// TwinCAT 3 PLC project PLC
// ProgramVersion: 3.1.4024.0
// CompilerDefines: MachineB
// libraries:
//   Tc2_Standard, * (Beckhoff Automation GmbH)
//   Tc2_System, * (Beckhoff Automation GmbH)
//   Tc3_Module, * (Beckhoff Automation GmbH)
// project tree:
//   Base/Datatype/ ST_Result.TcDUT
//   Base/FunctionBlock/ FB_Command.TcPOU
//   Base/Interface/ IBase.TcIO, ICommand.TcIO, IResult.TcIO
//   InterfaceBasics/DisplayExample/ FB_Display.TcPOU, FB_ProgressBar.TcPOU, IDisplay.TcIO
//   InterfaceBasics/SequenceExample/ FB_CylinderDoubleActing.TcPOU (not stored), FB_CylinderSequence.TcPOU, FB_CylinderSpringReturn.TcPOU (not stored), ICylinder.TcIO
//   InterfaceBasics/ PrgInterfaceBasics.TcPOU
//   / MAIN.TcPOU, PlcTask.TcTTO
// real-time tasks:
//   TASK PlcTask: cycle T#10ms, priority 20, ADS port 350

CONFIGURATION PLC
    RESOURCE PLC ON TwinCAT3
        TASK PlcTask(INTERVAL := T#10ms, PRIORITY := 20);
        PROGRAM MAIN WITH PlcTask : MAIN;
    END_RESOURCE
END_CONFIGURATION

// ---- Base/Datatype/ST_Result.TcDUT
{attribute 'pack_mode' := '1'}
TYPE ST_Result :
	STRUCT
		Busy	: BOOL;
		Error	: BOOL;
		Done	: BOOL;
		ErrorId : DINT;
	END_STRUCT
END_TYPE

// ---- Base/Interface/IBase.TcIO
INTERFACE IBase EXTENDS __System.IQueryInterface

END_INTERFACE

// ---- Base/Interface/ICommand.TcIO
INTERFACE ICommand EXTENDS IResult

PROPERTY Sequence : DINT
GET
END_GET
SET
END_SET
END_PROPERTY

METHOD Start : ICommand
VAR_INPUT
END_VAR
END_METHOD

END_INTERFACE

// ---- Base/Interface/IResult.TcIO
INTERFACE IResult EXTENDS __SYSTEM.IQueryInterface

PROPERTY Busy : BOOL
GET
END_GET
SET
END_SET
END_PROPERTY

PROPERTY Done : BOOL
GET
END_GET
SET
END_SET
END_PROPERTY

PROPERTY Error : BOOL
GET
END_GET
SET
END_SET
END_PROPERTY

PROPERTY ErrorId : DINT
GET
END_GET
SET
END_SET
END_PROPERTY

END_INTERFACE

// ---- InterfaceBasics/DisplayExample/IDisplay.TcIO
INTERFACE IDisplay EXTENDS IBase

METHOD Show : BOOL
VAR_INPUT
	Message : T_MaxString;
END_VAR
END_METHOD

END_INTERFACE

// ---- InterfaceBasics/SequenceExample/ICylinder.TcIO
INTERFACE ICylinder EXTENDS IBase

METHOD Extend : BOOL
VAR_INPUT
END_VAR
END_METHOD

METHOD Retract : BOOL
VAR_INPUT
END_VAR
END_METHOD

END_INTERFACE

// ---- MAIN.TcPOU
PROGRAM MAIN
VAR
END_VAR

PrgInterfaceBasics();

END_PROGRAM

// ---- InterfaceBasics/PrgInterfaceBasics.TcPOU
PROGRAM PrgInterfaceBasics
VAR
	// Interface Sequence Example
	{IF defined (MachineA)}
	CylinderSpringReturn : FB_CylinderSpringReturn;
	{ELSE}
	CylinderDoubleActing : FB_CylinderDoubleActing;
	{END_IF}
	CylinderSequence : FB_CylinderSequence;

	// Interface Display Example
	Display		 : FB_Display;
	ProgressBar	 : FB_ProgressBar;
	MainSequence : DINT := 0;
END_VAR

// Interface Sequence Example
{IF defined (MachineA)}

// Run Sequence with first Cylinder Type
CylinderSequence.Run(Cylinder := CylinderSpringReturn);
{ELSE}
CASE MainSequence OF
	0:
		IF CylinderSequence.Run(Cylinder := CylinderDoubleActing).Start().Busy THEN
			MainSequence := MainSequence + 10;
		END_IF

	10:
		IF CylinderSequence.Run(Cylinder := CylinderDoubleActing).Done THEN
			MainSequence := MainSequence + 10;
		END_IF

	20: // Next Command
END_CASE

{END_IF}

// Interface Display Example
ProgressBar.DisplayProgress(Display);

END_PROGRAM

// ---- InterfaceBasics/SequenceExample/FB_CylinderSequence.TcPOU
FUNCTION_BLOCK FB_CylinderSequence
VAR
	
END_VAR

METHOD PUBLIC Run : ICommand
VAR_INPUT
	Cylinder : ICylinder;
END_VAR

VAR_INST
	WaitTime : TON;
	Command	 : FB_Command;
END_VAR
IF Cylinder = 0 THEN
	Command.Error	:= TRUE;
	Command.ErrorId := 1;
	RETURN;
END_IF

CASE Command.Sequence OF
	0: // Extend
		IF Cylinder.Extend() THEN
			Command.Sequence := Command.Sequence + 10;
		END_IF

	10: // Wait 1s
		WaitTime.IN := TRUE;
		IF WaitTime.Q THEN
			WaitTime.IN		 := FALSE;
			Command.Sequence := Command.Sequence + 10;
		END_IF

	20: // Retract
		IF Cylinder.Retract() THEN
			Command.Sequence := Command.Sequence + 10;
		END_IF

	30: // Wait 1s
		WaitTime.IN := TRUE;
		IF WaitTime.Q THEN
			WaitTime.IN		 := FALSE;
			Command.Sequence := Command.Sequence + 10;
		END_IF

	40: // Done
		Command.Busy := FALSE;
		Command.Done := TRUE;
END_CASE

WaitTime(PT := T#1S);
Run := Command;
END_METHOD

END_FUNCTION_BLOCK

// ---- Base/FunctionBlock/FB_Command.TcPOU
{attribute 'no_explicit_call' := 'Do not call this FB directly!'}
FUNCTION_BLOCK FB_Command IMPLEMENTS ICommand
VAR
	_Result		   : ST_Result;
	_SequenceState : DINT;
END_VAR

PROPERTY Busy : BOOL
GET
Busy := _Result.Busy;
END_GET
SET
_Result.Busy := Busy;
END_SET
END_PROPERTY

PROPERTY Done : BOOL
GET
Done := _Result.Done;
END_GET
SET
_Result.Done := Done;
END_SET
END_PROPERTY

PROPERTY Error : BOOL
GET
Error := _Result.Error;
END_GET
SET
_Result.Error := Error;
END_SET
END_PROPERTY

PROPERTY ErrorId : DINT
GET
ErrorId := _Result.ErrorId;
END_GET
SET
_Result.ErrorId := ErrorId;
END_SET
END_PROPERTY

PROPERTY Sequence : DINT
GET
Sequence := _SequenceState;
END_GET
SET
_SequenceState := Sequence;
END_SET
END_PROPERTY

METHOD Start : ICommand
VAR_INPUT
END_VAR
_SequenceState	:= 0;
_Result.Done	:= FALSE;
_Result.Busy	:= TRUE;
_Result.Error	:= FALSE;
_Result.ErrorId := 0;
Start			:= This^;
END_METHOD

END_FUNCTION_BLOCK

// ---- InterfaceBasics/DisplayExample/FB_Display.TcPOU
FUNCTION_BLOCK FB_Display IMPLEMENTS IDisplay
VAR
END_VAR

METHOD Show : BOOL
VAR_INPUT
	Message : T_MaxString;
END_VAR
ADSLOGSTR(msgCtrlMask := ADSLOG_MSGTYPE_LOG, msgFmtStr := '%s', strArg := Message);
END_METHOD

END_FUNCTION_BLOCK

// ---- InterfaceBasics/DisplayExample/FB_ProgressBar.TcPOU
FUNCTION_BLOCK FB_ProgressBar IMPLEMENTS IBase
VAR
END_VAR

METHOD DisplayProgress : BOOL
VAR_INPUT
	ipDisplay : IDisplay;
END_VAR

VAR_INST
	Progress : UINT;
END_VAR
IF ipDisplay = 0 THEN
	// Return if Display Type is invalid
	RETURN;
END_IF

CASE Progress OF
	0:
		ipDisplay.Show('0%');
		Progress := 10;

	10:
		ipDisplay.Show('10%');
		Progress := 50;

	50:
		ipDisplay.Show('50%');
		Progress := 99;

	99:
		ipDisplay.Show('99%');
		Progress := 100;

	100:
		ipDisplay.Show('100%');
		Progress := 101;
END_CASE
END_METHOD

END_FUNCTION_BLOCK
